FUNCTION_BLOCK CLSender (* Basic FB with empty ECC *)
  (* Standard: 61499-2 *)
  (* Version 1.0, 2020-10-21, chong *)
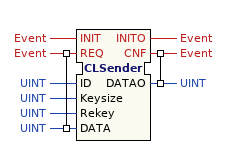
  EVENT_INPUT
    INIT;
    REQ WITH DATA;
  END_EVENT
  EVENT_OUTPUT
    INITO;
    CNF WITH DATAO;
  END_EVENT
  VAR_INPUT
    ID : UINT;
    Keysize : UINT;
    Rekey : UINT;
    DATA : UINT;
  END_VAR
  VAR_OUTPUT
    DATAO : UINT;
  END_VAR
  EC_STATES
    START; (* Initial State *)
  END_STATES
END_FUNCTION_BLOCK
